TYPE ST_GPS_OUTPUTS :
STRUCT
END_STRUCT
END_TYPE

(* stored: Version 1.1.0.1, ProductVersion 3.1.4022.11
   DUT ST_GPS_OUTPUTS: Id {51f41ddb-f135-4801-ae62-492150c4e245} *)
